ABB RAPID module: Module1.mod

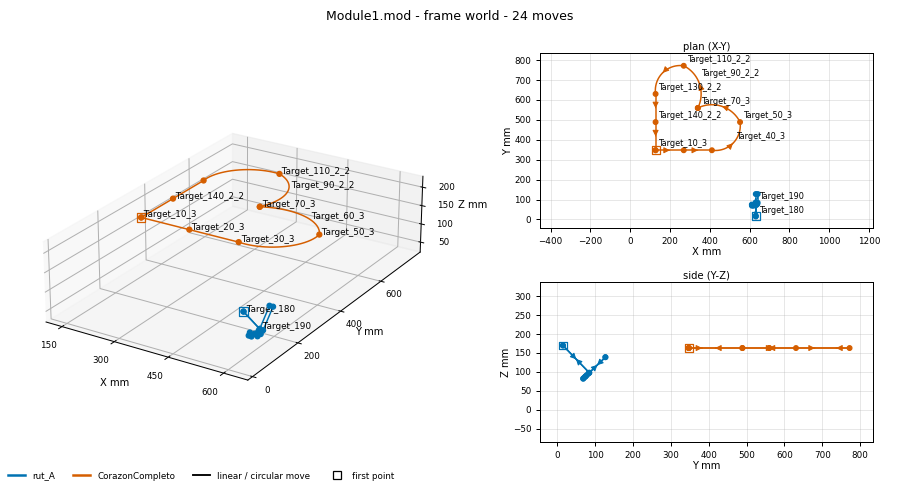
[picture p0: tool path of Module1.mod in frame world, 24 of 37 moves have a stored position in this frame; points joined in program order, loops and branches not executed]
MODULE Module1
    PERS string strOPC:= "timestamp";
    VAR bool bOPC :=TRUE;
    PERS bool bOPC2 :=TRUE;
    PERS num Cont :=90;

    PERS num IOTJ1 :=0;
    PERS num IOTJ2 :=1027;
    PERS num IOTJ3 :=926;
    PERS num IOTJ4 :=1018;
    PERS num IOTJ5 :=1021;
    PERS num IOTJ6 :=1025;

    PERS num POSX:=227.697;
    PERS num POSY:=520.922;
    PERS num POSZ:=729.274;

    PERS num MOVEPOSX:=5;
    PERS num MOVEPOSY:=1;
    PERS num MOVEPOSZ:=2;


    VAR robtarget posMoveL;
    VAR pos pos1;



    CONST jointtarget JointTarget_2:=[[0,50,-40,70,-50,-50],[9E+09,9E+09,9E+09,9E+09,9E+09,9E+09]];
    CONST jointtarget JointTarget_1:=[[0,20,-20,40,-20,-20],[9E+09,9E+09,9E+09,9E+09,9E+09,9E+09]];
    CONST jointtarget HomeP:=[[0,0,0,0,0,0],[9E+09,9E+09,9E+09,9E+09,9E+09,9E+09]];
    CONST jointtarget HomeR:=[[0,0,0,0,30,0],[9E+09,9E+09,9E+09,9E+09,9E+09,9E+09]];
    CONST jointtarget JointTarget_TL:=[[90,40,-45,0,0,0],[9E+09,9E+09,9E+09,9E+09,9E+09,9E+09]];
    CONST jointtarget JointTarget_TR:=[[-90,40,-45,0,0,0],[9E+09,9E+09,9E+09,9E+09,9E+09,9E+09]];
    !Init Vars cortadp
    CONST robtarget Home:=[[689.268487273,0,537.14730631],[0.190808996,0,0.981627183,0],[0,0,0,0],[9E+09,9E+09,9E+09,9E+09,9E+09,9E+09]];
    CONST robtarget Target_10:=[[800,100,300],[0,0,1,0],[0,0,0,0],[9E+09,9E+09,9E+09,9E+09,9E+09,9E+09]];
    CONST robtarget Target_20:=[[500,100,300],[0,0,1,0],[0,-1,0,0],[9E+09,9E+09,9E+09,9E+09,9E+09,9E+09]];
    PERS intnum veces;
    CONST robtarget Target_30:=[[500,400,300],[0,0,1,0],[0,-1,0,0],[9E+09,9E+09,9E+09,9E+09,9E+09,9E+09]];
    CONST robtarget Target_40:=[[800,400,300],[0,0,1,0],[0,-1,0,0],[9E+09,9E+09,9E+09,9E+09,9E+09,9E+09]];
    CONST robtarget Target_50:=[[800,-250,300],[0,0,1,0],[0,0,0,0],[9E+09,9E+09,9E+09,9E+09,9E+09,9E+09]];
    CONST robtarget Target_70:=[[500,-250,300],[0,0,1,0],[-1,0,-1,0],[9E+09,9E+09,9E+09,9E+09,9E+09,9E+09]];
    CONST robtarget Centro:=[[650,-250,403.186020656],[0,0,1,0],[-1,0,-1,0],[9E+09,9E+09,9E+09,9E+09,9E+09,9E+09]];
    CONST robtarget Target_80:=[[650,-100,300],[0,0,1,0],[-1,0,-1,0],[9E+09,9E+09,9E+09,9E+09,9E+09,9E+09]];
    CONST robtarget Target_60:=[[650,-400,300],[0,0,1,0],[-1,0,-1,0],[9E+09,9E+09,9E+09,9E+09,9E+09,9E+09]];
    CONST robtarget Target_120:=[[800,-100,300],[0,0,1,0],[-1,0,-1,0],[9E+09,9E+09,9E+09,9E+09,9E+09,9E+09]];
    CONST robtarget Target_100:=[[500,-400,300],[0,0,1,0],[-1,0,-1,0],[9E+09,9E+09,9E+09,9E+09,9E+09,9E+09]];
    CONST robtarget Target_90:=[[800,-400,300],[0,0,1,0],[-1,0,-1,0],[9E+09,9E+09,9E+09,9E+09,9E+09,9E+09]];
    CONST robtarget Target_110:=[[500,-100,300],[0,0,1,0],[-1,0,-1,0],[9E+09,9E+09,9E+09,9E+09,9E+09,9E+09]];
    !Fin Vars cortadp



    !Inicio Vars corazon
    CONST robtarget Target_10_3:=[[350,0,0],[0.707106781,0,0.707106781,0],[0,0,0,1],[9E+09,9E+09,9E+09,9E+09,9E+09,9E+09]];
    CONST robtarget Target_20_3:=[[450,-100,0],[0.707106781,0,0.707106781,0],[-1,-1,0,1],[9E+09,9E+09,9E+09,9E+09,9E+09,9E+09]];
    CONST robtarget Target_30_3:=[[550,-200,0],[0.707106781,0,0.707106781,0],[-1,-1,0,1],[9E+09,9E+09,9E+09,9E+09,9E+09,9E+09]];
    CONST robtarget Target_40_3:=[[650,-250,0],[0.707106781,0,0.707106781,0],[-1,-1,0,1],[9E+09,9E+09,9E+09,9E+09,9E+09,9E+09]];
    CONST robtarget Target_50_3:=[[750,-200,0],[0.707106781,0,0.707106781,0],[-1,-1,0,1],[9E+09,9E+09,9E+09,9E+09,9E+09,9E+09]];
    CONST robtarget Target_60_3:=[[750,-100,0],[0.707106781,0,0.707106781,0],[-1,-1,0,1],[9E+09,9E+09,9E+09,9E+09,9E+09,9E+09]];
    CONST robtarget Target_70_3:=[[650,0,0],[0.707106781,0,0.707106781,0],[0,0,0,1],[9E+09,9E+09,9E+09,9E+09,9E+09,9E+09]];
    CONST robtarget Target_80_2_2:=[[650,0,0],[0.707106781,0,0.707106781,0],[0,0,0,1],[9E+09,9E+09,9E+09,9E+09,9E+09,9E+09]];
    CONST robtarget Target_90_2_2:=[[750,100,0],[0.707106781,0,0.707106781,0],[-1,-1,0,1],[9E+09,9E+09,9E+09,9E+09,9E+09,9E+09]];
    CONST robtarget Target_110_2_2:=[[750,200,0],[0.707106781,0,0.707106781,0],[0,0,-1,1],[9E+09,9E+09,9E+09,9E+09,9E+09,9E+09]];
    CONST robtarget Target_120_2_2:=[[650,250,0],[0.707106781,0,0.707106781,0],[0,0,-1,1],[9E+09,9E+09,9E+09,9E+09,9E+09,9E+09]];
    CONST robtarget Target_130_2_2:=[[550,200,0],[0.707106781,0,0.707106781,0],[0,0,-1,1],[9E+09,9E+09,9E+09,9E+09,9E+09,9E+09]];
    CONST robtarget Target_140_2_2:=[[450,100,0],[0.707106781,0,0.707106781,0],[0,0,0,1],[9E+09,9E+09,9E+09,9E+09,9E+09,9E+09]];
    CONST robtarget Target_1010_2_2:=[[350,0,0],[0.707106781,0,0.707106781,0],[0,0,0,1],[9E+09,9E+09,9E+09,9E+09,9E+09,9E+09]];
    CONST robtarget home_2:=[[506.292,0,679.5],[0.5,0,0.866025404,0],[0,-2,-2,1],[9E+09,9E+09,9E+09,9E+09,9E+09,9E+09]];
    !Fin Vars corazon

    !Inicio vars A
    CONST robtarget Target_180:=[[-130.684278975,166.513773343,100.000300403],[-0.000000024,0.819152044,-0.573576437,-0.000000024],[0,1,-1,1],[9E+09,9E+09,9E+09,9E+09,9E+09,9E+09]];
    CONST robtarget Target_190:=[[-130.684278975,166.513780154,0.000300403],[0.000000024,-0.707106781,0.707106781,0.000000024],[0,1,-1,1],[9E+09,9E+09,9E+09,9E+09,9E+09,9E+09]];
    CONST robtarget Target_200:=[[-130.684278975,107.401152167,0.000296377],[0.000000024,-0.707106781,0.707106781,0.000000024],[0,1,-1,1],[9E+09,9E+09,9E+09,9E+09,9E+09,9E+09]];
    CONST robtarget Target_210:=[[-140.172333582,107.401152167,0.000296377],[0.000000024,-0.707106781,0.707106781,0.000000024],[0,1,-1,1],[9E+09,9E+09,9E+09,9E+09,9E+09,9E+09]];
    CONST robtarget Target_220:=[[-140.172333582,167.537670939,0.000300473],[0.000000024,0.819152044,-0.573576437,-0.000000024],[0,1,-1,1],[9E+09,9E+09,9E+09,9E+09,9E+09,9E+09]];
    CONST robtarget Target_230:=[[-138.363459862,177.588865478,0.000301158],[0.000000024,0.819152044,-0.573576437,-0.000000024],[0,1,-1,1],[9E+09,9E+09,9E+09,9E+09,9E+09,9E+09]];
    CONST robtarget Target_240:=[[-132.936838702,184.67077674,0.00030164],[0.000000024,0.819152044,-0.573576437,-0.000000024],[0,1,-1,1],[9E+09,9E+09,9E+09,9E+09,9E+09,9E+09]];
    CONST robtarget Target_250:=[[-118.807145869,188.971118037,0.000301932],[0.000000024,-0.707106781,0.707106781,0.000000024],[0,1,-1,1],[9E+09,9E+09,9E+09,9E+09,9E+09,9E+09]];
    CONST robtarget Target_260:=[[-111.23035406,188.561561724,0.000301905],[0.000000024,-0.707106781,0.707106781,0.000000024],[0,1,-1,1],[9E+09,9E+09,9E+09,9E+09,9E+09,9E+09]];
    CONST robtarget Target_270:=[[-110.820797746,180.779991758,0.000301375],[0.000000024,-0.707106781,0.707106781,0.000000024],[0,1,-1,1],[9E+09,9E+09,9E+09,9E+09,9E+09,9E+09]];
    CONST robtarget Target_280:=[[-123.482913787,180.353370597,0.000301346],[0.000000024,-0.707106781,0.707106781,0.000000024],[0,1,-1,1],[9E+09,9E+09,9E+09,9E+09,9E+09,9E+09]];
    CONST robtarget Target_290:=[[-129.882231193,172.605930324,0.000300819],[0.000000024,-0.707106781,0.707106781,0.000000024],[0,1,-1,1],[9E+09,9E+09,9E+09,9E+09,9E+09,9E+09]];
    CONST robtarget Target_300:=[[-130.684278975,166.513780154,0.000300403],[0.000000024,-0.707106781,0.707106781,0.000000024],[0,1,-1,1],[9E+09,9E+09,9E+09,9E+09,9E+09,9E+09]];
    CONST robtarget Target_310:=[[-130.684278975,166.513773343,100.000300403],[0.000000024,0.819152044,-0.573576437,-0.000000024],[0,1,-1,1],[9E+09,9E+09,9E+09,9E+09,9E+09,9E+09]];

    !Fin Vars A


    VAR jointtarget myJointTarget;
    PROC main()
        ActualizarDatoPos;
        SETDO DO_IOT_01,1;
        WaitDI DI_IOT_02,1;
        WaitDI DI_IOT_01,1;
        WaitDI DI_IOT_02,1;
        SETDO DO_IOT_01,0;
        TEST DI_INT_IOT_01

            CASE 1:
                ToHomeP;
            CASE 2:
                ToHomeR;
            CASE 3:
                ToolQL;
            CASE 4:
                ToolQR;
            CASE 5:
                Security;
            CASE 6:
                MoveProcJInt;
            CASE 7:
                MovePosLInt;
            CASE 8:
                CortadoFull;
            CASE 9:
                CorazonCompleto;
            CASE 10:
                rut_A;
        ENDTEST

    ENDPROC
    PROC ToHomeP()
        ActualizarDatoPos;
        MoveAbsJ HomeP,v100,z10,ToolAJATCP\WObj:=WOAJA;
    ENDPROC

    PROC ToHomeR()
        ActualizarDatoPos;
        MoveAbsJ HomeR,v100,z10,ToolAJATCP\WObj:=WOAJA;
    ENDPROC


    PROC Security()
        ActualizarDatoPos;
        MoveAbsJ HomeP,v100,z10,ToolAJATCP\WObj:=WOAJA;
        ActualizarDatoPos;
        MoveAbsJ JointTarget_1,v100,z10,ToolAJATCP\WObj:=WOAJA;
        ActualizarDatoPos;
        MoveAbsJ JointTarget_2,v100,z10,ToolAJATCP\WObj:=WOAJA;
    ENDPROC
    PROC ToolQL()
        MoveAbsJ HomeP,v100,z10,ToolAJATCP\WObj:=WOAJA;
        ActualizarDatoPos;
        MoveAbsJ JointTarget_TL,v100,z10,ToolAJATCP\WObj:=WOAJA;
    ENDPROC

    PROC ToolQR()
        ActualizarDatoPos;
        MoveAbsJ HomeP,v100,z10,ToolAJATCP\WObj:=WOAJA;
        ActualizarDatoPos;
        MoveAbsJ JointTarget_TR,v100,z10,ToolAJATCP\WObj:=WOAJA;
    ENDPROC
    PROC rut_A()
        MoveL Target_180,v100,z10,ToolAJATCP\WObj:=WOAJA;
        MoveL Target_190,v100,z10,ToolAJATCP\WObj:=WOAJA;
        MoveL Target_200,v100,z10,ToolAJATCP\WObj:=WOAJA;
        MoveL Target_210,v100,z10,ToolAJATCP\WObj:=WOAJA;
        MoveL Target_220,v100,z10,ToolAJATCP\WObj:=WOAJA;
        MoveL Target_230,v100,z10,ToolAJATCP\WObj:=WOAJA;
        MoveL Target_240,v100,z10,ToolAJATCP\WObj:=WOAJA;
        MoveL Target_250,v100,z10,ToolAJATCP\WObj:=WOAJA;
        MoveL Target_260,v100,z10,ToolAJATCP\WObj:=WOAJA;
        MoveL Target_270,v100,z10,ToolAJATCP\WObj:=WOAJA;
        MoveL Target_280,v100,z10,ToolAJATCP\WObj:=WOAJA;
        MoveL Target_290,v100,z10,ToolAJATCP\WObj:=WOAJA;
        MoveL Target_300,v100,z10,ToolAJATCP\WObj:=WOAJA;
        MoveL Target_310,v100,z10,ToolAJATCP\WObj:=WOAJA;
    ENDPROC



    PROC ActualizarDatoPos()
        pos1 := CPos(\Tool:=tool0 \WObj:=wobj0);
        POSX:=pos1.x;
        POSY:=pos1.y;
        POSZ:=pos1.z;
    ENDPROC


    PROC MoveProcJ()
        myJointTarget := [[IOTJ1,IOTJ2,IOTJ3,IOTJ4,IOTJ5,IOTJ6],[9E+09,9E+09,9E+09,9E+09,9E+09,9E+09]];
        MoveAbsJ myJointTarget,v100,z10,ToolAJATCP\WObj:=WOAJA;
    ENDPROC

    PROC MoveProcJInt()
        !IOTJ1:=DINT_J1-1000;
        myJointTarget := [[DINT_J1-1000,DINT_J2-1000,DINT_J3-1000,DINT_J4-1000,DINT_J5-1000,DINT_J6-1000],[9E+09,9E+09,9E+09,9E+09,9E+09,9E+09]];
        MoveAbsJ myJointTarget,v100,z10,ToolAJATCP\WObj:=WOAJA;
    ENDPROC


    PROC MovePosL()
        posMoveL:=CRobT(\Tool:=tool0 \WObj:=wobj0);
        posMoveL.trans.x:=posMoveL.trans.x+MOVEPOSX;
        posMoveL.trans.y:=posMoveL.trans.y+MOVEPOSY;
        posMoveL.trans.z:=posMoveL.trans.z+MOVEPOSZ;
        MoveL posMoveL,v50,z5,tool0\WObj:=wobj0;
    ENDPROC

    PROC MovePosLInt()
        posMoveL:=CRobT(\Tool:=tool0 \WObj:=wobj0);
        posMoveL.trans.x:=posMoveL.trans.x+DINT_MX-1000;
        posMoveL.trans.y:=posMoveL.trans.y+DINT_MY-1000;
        posMoveL.trans.z:=posMoveL.trans.z+DINT_MZ-1000;
        MoveL posMoveL,v50,z5,tool0\WObj:=wobj0;
    ENDPROC

    PROC CortadoFull()
        Pegado;
        ToHomeR;
        ToHomeR;
        Cortado;
    ENDPROC

    PROC Pegado()
        !MoveJ Target_10,v200,fine,MyTool\WObj:=Workobject_1;
        !MoveJ Target_20,v200,fine,MyTool\WObj:=Workobject_1;
        !MoveJ Target_30,v200,fine,MyTool\WObj:=Workobject_1;
        !MoveJ Target_40,v200,fine,MyTool\WObj:=Workobject_1;
        !MoveJ Target_10,v200,fine,MyTool\WObj:=Workobject_1;
    ENDPROC
    PROC Cortado()
        !MoveJ Target_50,v200,fine,MyTool\WObj:=Workobject_2;
        !MoveJ Target_70,v200,fine,MyTool\WObj:=Workobject_2;
        !MoveJ Centro,v200,fine,MyTool\WObj:=Workobject_2;
        !MoveJ Target_80,v200,fine,MyTool\WObj:=Workobject_2;
        !MoveJ Target_60,v200,fine,MyTool\WObj:=Workobject_2;
        !MoveJ Centro,v200,fine,MyTool\WObj:=Workobject_2;
        !MoveJ Target_120,v200,fine,MyTool\WObj:=Workobject_2;
        !MoveJ Target_100,v200,fine,MyTool\WObj:=Workobject_2;
        !MoveJ Centro,v200,fine,MyTool\WObj:=Workobject_2;
        !MoveJ Target_90,v200,fine,MyTool\WObj:=Workobject_2;
        !MoveJ Target_110,v200,fine,MyTool\WObj:=Workobject_2;
        !MoveJ Centro,v200,fine,MyTool\WObj:=Workobject_2;
    ENDPROC

PROC CorazonCompleto()
        MoveJ Target_10_3,v200,z5,tool0\WObj:=MiMarcoDeCorazon;
        MoveL Target_20_3,v200,z5,tool0\WObj:=MiMarcoDeCorazon;
        MoveL Target_30_3,v200,z5,tool0\WObj:=MiMarcoDeCorazon;
        MoveC Target_40_3,Target_50_3,v200,z5,tool0\WObj:=MiMarcoDeCorazon;
        MoveC Target_60_3,Target_70_3,v200,z5,tool0\WObj:=MiMarcoDeCorazon;
        MoveL Target_80_2_2,v200,z5,tool0\WObj:=MiMarcoDeCorazon;
        MoveC Target_90_2_2,Target_110_2_2,v200,z5,tool0\WObj:=MiMarcoDeCorazon;
        MoveC Target_120_2_2,Target_130_2_2,v200,z5,tool0\WObj:=MiMarcoDeCorazon;
        MoveL Target_140_2_2,v200,z5,tool0\WObj:=MiMarcoDeCorazon;
        MoveL Target_1010_2_2,v200,z5,tool0\WObj:=MiMarcoDeCorazon;
        ToHomeR;
    ENDPROC
ENDMODULE
